Fanuc KAREL source: FanucPortOpenTest.kl

PROGRAM FANUC_PORT_OPEN_TEST
%NOLOCKGROUP
%NOPAUSE = ERROR + COMMAND + TPENABLE
%COMMENT = 'Open S4 TCP server port test'
%ENVIRONMENT sysdef
%ENVIRONMENT fdev
%ENVIRONMENT flbt

VAR
  channel : FILE
  status  : INTEGER
  entry   : INTEGER
  cmd     : STRING[254]
  session_on : BOOLEAN

BEGIN
  SET_FILE_ATR(channel, ATR_IA)

  -- S4 maps to $HOSTS_CFG[4]. PC should connect to robot_ip:9000.
  SET_VAR(entry, '*SYSTEM*', '$HOSTS_CFG[4].$SERVER_PORT', 9000, status)
  WRITE('SET S4 PORT STATUS=', status, CR)

  MSG_CONNECT('S4:', status)
  WRITE('MSG_CONNECT S4 STATUS=', status, CR)
  IF status <> 0 THEN
    ABORT
  ENDIF

  WRITE('Waiting for TCP client on S4 port 9000...', CR)

  OPEN FILE channel('rw', 'S4:')
  status = IO_STATUS(channel)
  WRITE('OPEN S4 STATUS=', status, CR)

  IF status = 0 THEN
    WRITE channel('OK:PORT_OPEN', CR)
    session_on = TRUE

    WHILE session_on DO
      BYTES_AHEAD(channel, entry, status)
      IF status <> 0 THEN
        session_on = FALSE
      ELSE
        IF entry > 0 THEN
          READ channel(cmd)
          status = IO_STATUS(channel)
          IF status <> 0 THEN
            session_on = FALSE
          ELSE
            IF cmd = 'HELLO' THEN
              WRITE channel('OK:HELLO', CR)
            ELSE
              IF cmd = 'QUIT' THEN
                WRITE channel('OK:QUIT', CR)
                session_on = FALSE
              ELSE
                WRITE channel('ECHO:', cmd, CR)
              ENDIF
            ENDIF
          ENDIF
        ENDIF
      ENDIF
    ENDWHILE

    CLOSE FILE channel
    WRITE('Client disconnected, S4 file closed', CR)
  ENDIF

  MSG_DISCO('S4:', status)
  WRITE('MSG_DISCO S4 STATUS=', status, CR)
END FANUC_PORT_OPEN_TEST
